(* IEC 61131-3 sources: RL_MAR/experiments/comparison/llm4plc/results/gpt-4o-mini_20260506_100619/20260506_101548, 1 file *)

(* ---- generated_code_iteration_0.st ---- *)
ructured-text
FUNCTION_BLOCK FlowerArrangingMachine
VAR_INPUT
    FlowerTypeSensor : INT; (* Input for detecting flower type *)
    FlowerColorSensor : INT; (* Input for detecting flower color *)
END_VAR
VAR_OUTPUT
    ArrangingMechanism : INT; (* Output for controlling arranging mechanism *)
    ConveyorBelt : BOOL; (* Output for controlling conveyor belt *)
END_VAR

VAR
    (* State declaration *)
    CurrentState : INT := 0; (* 0: INITIALIZE, 1: DETERMINE_ARRANGING_MECHANISM *)
END_VAR

(* Main control logic *)
CASE CurrentState OF
    0: (* INITIALIZE state *)
        ArrangingMechanism := 0;
        ConveyorBelt := FALSE;
        CurrentState := 1; (* Transition to DETERMINE_ARRANGING_MECHANISM state *)

    1: (* DETERMINE_ARRANGING_MECHANISM state *)
        IF FlowerTypeSensor = 1 AND FlowerColorSensor = 1 THEN
            ArrangingMechanism := 1; (* Red type 1 flower *)
        ELSIF FlowerTypeSensor = 1 AND FlowerColorSensor = 2 THEN
            ArrangingMechanism := 2; (* Blue type 1 flower *)
        ELSIF FlowerTypeSensor = 2 AND FlowerColorSensor = 1 THEN
            ArrangingMechanism := 3; (* Red type 2 flower *)
        ELSIF FlowerTypeSensor = 2 AND FlowerColorSensor = 2 THEN
            ArrangingMechanism := 4; (* Blue type 2 flower *)
        ELSE
            ArrangingMechanism := 0; (* Any other combination *)
        END_IF;

        IF ArrangingMechanism <> 0 THEN
            ConveyorBelt := TRUE; (* Activate conveyor belt *)
        ELSE
            ConveyorBelt := FALSE; (* Deactivate conveyor belt *)
        END_IF;

        (* Remain in DETERMINE_ARRANGING_MECHANISM state for next cycle *)
END_CASE

END_FUNCTION_BLOCK
